PROGRAM AxisAllCtrl
VAR
	i				:USINT := 1;

END_VAR



//所有Axis上电
IF bAxis_All_Enable THEN
	FOR i:=1 TO nAxisNum DO
		aAxis_All_Enable_Group[i]^:=TRUE;
	END_FOR
END_IF

//所有Axis下电
IF bAxis_All_Disable THEN
	FOR i:=1 TO nAxisNum DO
		aAxis_All_Enable_Group[i]^:=FALSE;
	END_FOR
END_IF

//所有轴清除故障
IF bAxis_All_Reset THEN
	FOR i:=1 TO nAxisNum DO
		aAxis_All_Reset_Group[i]^:=TRUE;
	END_FOR
ELSE
	FOR i:=1 TO nAxisNum DO
		aAxis_All_Reset_Group[i]^:=FALSE;
	END_FOR	
END_IF

END_PROGRAM

(* stored: Version 1.1.0.1, ProductVersion 3.1.4024.14
   POU AxisAllCtrl: Id {d3660b0b-86b3-46ef-a236-dea2cee54968}, SpecialFunc None *)
